LIN {X 0,Y 100.237,Z 319.477,A -85,B 0,C 180,E1 -28284.878,E2 -28284.878} C_VEL
LIN {X 0,Y 100.973,Z 322.725,A -85,B 0,C 180,E1 -28289.159,E2 -28289.159} C_VEL
LIN {X 0,Y 101.731,Z 327.087,A -85,B 0,C 180,E1 -28293.993,E2 -28293.993} C_VEL
LIN {X 0,Y 102.226,Z 331.393,A -85,B 0,C 180,E1 -28298.225,E2 -28298.225} C_VEL
LIN {X 0,Y 102.183,Z 334.397,A -85,B 0,C 180,E1 -28300.829,E2 -28300.829} C_VEL
LIN {X 0,Y 101.856,Z 336.169,A -85,B 0,C 180,E1 -28302.111,E2 -28302.111} C_VEL
LIN {X 0,Y 101.066,Z 337.874,A -85,B 0,C 180,E1 -28303.092,E2 -28303.092} C_VEL
LIN {X 0,Y 94.071,Z 347.385,A -85,B 0,C 180,E1 -28307.74,E2 -28307.74} C_VEL
LIN {X 0,Y 87.576,Z 355.164,A -85,B 0,C 180,E1 -28313.275,E2 -28313.275} C_VEL
LIN {X 0,Y 82.169,Z 361.026,A -85,B 0,C 180,E1 -28319.116,E2 -28319.116} C_VEL
LIN {X 0,Y 77.494,Z 365.857,A -85,B 0,C 180,E1 -28325.906,E2 -28325.906} C_VEL
LIN {X 0,Y 73.914,Z 369.582,A -85,B 0,C 180,E1 -28333.418,E2 -28333.418} C_VEL
LIN {X 0,Y 72.209,Z 371.5,A -85,B 0,C 180,E1 -28338.75,E2 -28338.75} C_VEL
LIN {X 0,Y 70.595,Z 372.917,A -85,B 0,C 180,E1 -28343.171,E2 -28343.171} C_VEL
LIN {X 0,Y 68.413,Z 374.026,A -85,B 0,C 180,E1 -28347.646,E2 -28347.646} C_VEL
LIN {X 0,Y 64.554,Z 375.318,A -85,B 0,C 180,E1 -28357.388,E2 -28357.388} C_VEL
LIN {X 0,Y 64.037,Z 375.526,A -85,B 0,C 180,E1 -28362.692,E2 -28362.692} C_VEL
LIN {X 0,Y 64.223,Z 375.507,A -85,B 0,C 180,E1 -28364.464,E2 -28364.464} C_VEL
LIN {X 0,Y 66.935,Z 374.948,A -85,B 0,C 180,E1 -28374.824,E2 -28374.824} C_VEL
LIN {X 0,Y 72.356,Z 372.767,A -85,B 0,C 180,E1 -28385.636,E2 -28385.636} C_VEL
LIN {X 0,Y 77.872,Z 370.014,A -85,B 0,C 180,E1 -28392.59,E2 -28392.59} C_VEL
LIN {X 0,Y 84.271,Z 366.237,A -85,B 0,C 180,E1 -28398.63,E2 -28398.63} C_VEL
LIN {X 0,Y 91.429,Z 361.324,A -85,B 0,C 180,E1 -28403.804,E2 -28403.804} C_VEL
LIN {X 0,Y 99.192,Z 355.123,A -85,B 0,C 180,E1 -28408.225,E2 -28408.225} C_VEL
LIN {X 0,Y 103.769,Z 350.924,A -85,B 0,C 180,E1 -28410.467,E2 -28410.467} C_VEL
LIN {X 0,Y 104.812,Z 347.909,A -85,B 0,C 180,E1 -28414.16,E2 -28414.16} C_VEL
LIN {X 0,Y 105.601,Z 344.619,A -85,B 0,C 180,E1 -28418.69,E2 -28418.69} C_VEL
LIN {X 0,Y 105.994,Z 341.263,A -85,B 0,C 180,E1 -28424.619,E2 -28424.619} C_VEL
LIN {X 0,Y 106.042,Z 339.662,A -85,B 0,C 180,E1 -28428.531,E2 -28428.531} C_VEL
LIN {X 0,Y 106.187,Z 338.276,A -85,B 0,C 180,E1 -28433.059,E2 -28433.059} C_VEL
LIN {X 0,Y 106.837,Z 336.92,A -85,B 0,C 180,E1 -28440,E2 -28440} C_VEL
LIN {X 0,Y 105.925,Z 338.695,A -85,B 0,C 180,E1 -28445.656,E2 -28445.656} C_VEL
LIN {X 0,Y 105.423,Z 341.22,A -85,B 0,C 180,E1 -28451.536,E2 -28451.536} C_VEL
LIN {X 0,Y 105.037,Z 343.497,A -85,B 0,C 180,E1 -28455.523,E2 -28455.523} C_VEL
LIN {X 0,Y 104.468,Z 346.468,A -85,B 0,C 180,E1 -28459.656,E2 -28459.656} C_VEL
LIN {X 0,Y 103.329,Z 351.55,A -85,B 0,C 180,E1 -28465.77,E2 -28465.77} C_VEL
LIN {X 0,Y 102.94,Z 353.062,A -85,B 0,C 180,E1 -28467.447,E2 -28467.447} C_VEL
LIN {X 0,Y 101.965,Z 354.793,A -85,B 0,C 180,E1 -28468.847,E2 -28468.847} C_VEL
LIN {X 0,Y 96.86,Z 361.172,A -85,B 0,C 180,E1 -28473.456,E2 -28473.456} C_VEL
LIN {X 0,Y 94.423,Z 363.454,A -85,B 0,C 180,E1 -28475.052,E2 -28475.052} C_VEL
LIN {X 0,Y 86.797,Z 369.418,A -85,B 0,C 180,E1 -28479.727,E2 -28479.727} C_VEL
LIN {X 0,Y 79.888,Z 374.149,A -85,B 0,C 180,E1 -28485.279,E2 -28485.279} C_VEL
LIN {X 0,Y 73.847,Z 377.783,A -85,B 0,C 180,E1 -28491.796,E2 -28491.796} C_VEL
LIN {X 0,Y 68.871,Z 380.421,A -85,B 0,C 180,E1 -28499.331,E2 -28499.331} C_VEL
LIN {X 0,Y 66.357,Z 381.688,A -85,B 0,C 180,E1 -28504.945,E2 -28504.945} C_VEL
LIN {X 0,Y 64.543,Z 382.528,A -85,B 0,C 180,E1 -28510.943,E2 -28510.943} C_VEL
LIN {X 0,Y 62.964,Z 383.019,A -85,B 0,C 180,E1 -28523.601,E2 -28523.601} C_VEL
LIN {X 0,Y 63.17,Z 382.685,A -85,B 0,C 180,E1 -28530.009,E2 -28530.009} C_VEL
LIN {X 0,Y 62.978,Z 381.865,A -85,B 0,C 180,E1 -28536.417,E2 -28536.417} C_VEL
LIN {X 0,Y 63.413,Z 380.607,A -85,B 0,C 180,E1 -28542.816,E2 -28542.816} C_VEL
LIN {X 0,Y 65.37,Z 377.946,A -85,B 0,C 180,E1 -28552.114,E2 -28552.114} C_VEL
LIN {X 0,Y 68.839,Z 374.259,A -85,B 0,C 180,E1 -28560.704,E2 -28560.704} C_VEL
LIN {X 0,Y 73.698,Z 369.456,A -85,B 0,C 180,E1 -28568.316,E2 -28568.316} C_VEL
LIN {X 0,Y 79.495,Z 363.369,A -85,B 0,C 180,E1 -28575.023,E2 -28575.023} C_VEL
LIN {X 0,Y 85.266,Z 357.204,A -85,B 0,C 180,E1 -28579.689,E2 -28579.689} C_VEL
LIN {X 0,Y 88.32,Z 352.824,A -85,B 0,C 180,E1 -28582.736,E2 -28582.736} C_VEL
LIN {X 0,Y 93.291,Z 344.019,A -85,B 0,C 180,E1 -28588.175,E2 -28588.175} C_VEL
LIN {X 0,Y 95.208,Z 339.981,A -85,B 0,C 180,E1 -28590.414,E2 -28590.414} C_VEL
LIN {X 0,Y 95.71,Z 338.033,A -85,B 0,C 180,E1 -28591.796,E2 -28591.796} C_VEL
LIN {X 0,Y 95.932,Z 333.079,A -85,B 0,C 180,E1 -28596.239,E2 -28596.239} C_VEL
LIN {X 0,Y 95.806,Z 327.088,A -85,B 0,C 180,E1 -28602.504,E2 -28602.504} C_VEL
LIN {X 0,Y 95.602,Z 323.433,A -85,B 0,C 180,E1 -28607.26,E2 -28607.26} C_VEL
LIN {X 0,Y 95.363,Z 320.851,A -85,B 0,C 180,E1 -28611.524,E2 -28611.524} C_VEL
LIN {X 0,Y 95.158,Z 319.066,A -85,B 0,C 180,E1 -28615.765,E2 -28615.765} C_VEL
LIN {X 0,Y 94.982,Z 318.072,A -85,B 0,C 180,E1 -28620.001,E2 -28620.001} C_VEL
LIN {X 0,Y 94.554,Z 318.54,A -85,B 0,C 180,E1 -28627.291,E2 -28627.291} C_VEL
LIN {X 0,Y 94.796,Z 319.647,A -85,B 0,C 180,E1 -28632.851,E2 -28632.851} C_VEL
LIN {X 0,Y 95.306,Z 322.239,A -85,B 0,C 180,E1 -28639.381,E2 -28639.381} C_VEL
LIN {X 0,Y 95.804,Z 324.716,A -85,B 0,C 180,E1 -28643.814,E2 -28643.814} C_VEL
LIN {X 0,Y 96.283,Z 328.257,A -85,B 0,C 180,E1 -28648.835,E2 -28648.835} C_VEL
LIN {X 0,Y 96.701,Z 332.759,A -85,B 0,C 180,E1 -28654.231,E2 -28654.231} C_VEL
LIN {X 0,Y 96.706,Z 336.521,A -85,B 0,C 180,E1 -28658.149,E2 -28658.149} C_VEL
LIN {X 0,Y 96.26,Z 338.595,A -85,B 0,C 180,E1 -28659.941,E2 -28659.941} C_VEL
LIN {X 0,Y 91.388,Z 345.102,A -85,B 0,C 180,E1 -28663.056,E2 -28663.056} C_VEL
LIN {X 0,Y 84.354,Z 353.212,A -85,B 0,C 180,E1 -28668.191,E2 -28668.191} C_VEL
LIN {X 0,Y 78.146,Z 359.73,A -85,B 0,C 180,E1 -28674.218,E2 -28674.218} C_VEL
LIN {X 0,Y 72.707,Z 364.935,A -85,B 0,C 180,E1 -28681.089,E2 -28681.089} C_VEL
LIN {X 0,Y 68.382,Z 368.985,A -85,B 0,C 180,E1 -28688.908,E2 -28688.908} C_VEL
LIN {X 0,Y 65.282,Z 372.001,A -85,B 0,C 180,E1 -28697.557,E2 -28697.557} C_VEL
LIN {X 0,Y 64.053,Z 373.495,A -85,B 0,C 180,E1 -28703.692,E2 -28703.692} C_VEL
LIN {X 0,Y 63.432,Z 375.223,A -85,B 0,C 180,E1 -28716.352,E2 -28716.352} C_VEL
LIN {X 0,Y 64.223,Z 375.507,A -85,B 0,C 180,E1 -28724.464,E2 -28724.464} C_VEL
LIN {X 0,Y 64.648,Z 375.451,A -85,B 0,C 180,E1 -28729.706,E2 -28729.706} C_VEL
LIN {X 0,Y 64.641,Z 374.849,A -85,B 0,C 180,E1 -28738.499,E2 -28738.499} C_VEL
LIN {X 0,Y 66.024,Z 373.597,A -85,B 0,C 180,E1 -28747.062,E2 -28747.062} C_VEL
LIN {X 0,Y 68.47,Z 372.339,A -85,B 0,C 180,E1 -28751.532,E2 -28751.532} C_VEL
LIN {X 0,Y 75.001,Z 369.204,A -85,B 0,C 180,E1 -28758.547,E2 -28758.547} C_VEL
LIN {X 0,Y 82.221,Z 365.031,A -85,B 0,C 180,E1 -28764.282,E2 -28764.282} C_VEL
LIN {X 0,Y 91.461,Z 358.667,A -85,B 0,C 180,E1 -28769.808,E2 -28769.808} C_VEL
LIN {X 0,Y 98.395,Z 352.93,A -85,B 0,C 180,E1 -28773.236,E2 -28773.236} C_VEL
LIN {X 0,Y 99.401,Z 350.464,A -85,B 0,C 180,E1 -28776.785,E2 -28776.785} C_VEL
LIN {X 0,Y 99.974,Z 348.824,A -85,B 0,C 180,E1 -28779.421,E2 -28779.421} C_VEL
LIN {X 0,Y 100.492,Z 346.577,A -85,B 0,C 180,E1 -28783.755,E2 -28783.755} C_VEL
LIN {X 0,Y 100.801,Z 344.873,A -85,B 0,C 180,E1 -28787.926,E2 -28787.926} C_VEL
LIN {X 0,Y 101.047,Z 343.664,A -85,B 0,C 180,E1 -28792.003,E2 -28792.003} C_VEL
LIN {X 0,Y 101.898,Z 342.177,A -85,B 0,C 180,E1 -28800,E2 -28800} C_VEL
LIN {X 0,Y 101.178,Z 343.307,A -85,B 0,C 180,E1 -28803.983,E2 -28803.983} C_VEL
LIN {X 0,Y 100.228,Z 346.059,A -85,B 0,C 180,E1 -28811.016,E2 -28811.016} C_VEL
LIN {X 0,Y 99.786,Z 347.751,A -85,B 0,C 180,E1 -28814.271,E2 -28814.271} C_VEL
LIN {X 0,Y 98.749,Z 351.134,A -85,B 0,C 180,E1 -28819.418,E2 -28819.418} C_VEL
LIN {X 0,Y 97.855,Z 354.006,A -85,B 0,C 180,E1 -28823.264,E2 -28823.264} C_VEL
LIN {X 0,Y 97.097,Z 355.997,A -85,B 0,C 180,E1 -28825.74,E2 -28825.74} C_VEL
LIN {X 0,Y 94.026,Z 359.653,A -85,B 0,C 180,E1 -28828.581,E2 -28828.581} C_VEL
LIN {X 0,Y 90.515,Z 363.192,A -85,B 0,C 180,E1 -28831.353,E2 -28831.353} C_VEL
LIN {X 0,Y 82.412,Z 369.123,A -85,B 0,C 180,E1 -28835.902,E2 -28835.902} C_VEL
LIN {X 0,Y 74.979,Z 373.826,A -85,B 0,C 180,E1 -28841.434,E2 -28841.434} C_VEL
LIN {X 0,Y 68.372,Z 377.433,A -85,B 0,C 180,E1 -28848.089,E2 -28848.089} C_VEL
LIN {X 0,Y 62.849,Z 380.046,A -85,B 0,C 180,E1 -28856.017,E2 -28856.017} C_VEL
LIN {X 0,Y 59.956,Z 381.297,A -85,B 0,C 180,E1 -28862.05,E2 -28862.05} C_VEL
LIN {X 0,Y 57.848,Z 382.116,A -85,B 0,C 180,E1 -28868.636,E2 -28868.636} C_VEL
LIN {X 0,Y 55.902,Z 382.584,A -85,B 0,C 180,E1 -28882.788,E2 -28882.788} C_VEL
LIN {X 0,Y 56.072,Z 382.239,A -85,B 0,C 180,E1 -28890.011,E2 -28890.011} C_VEL
LIN {X 0,Y 55.913,Z 381.394,A -85,B 0,C 180,E1 -28897.232,E2 -28897.232} C_VEL
LIN {X 0,Y 56.479,Z 380.123,A -85,B 0,C 180,E1 -28904.421,E2 -28904.421} C_VEL
LIN {X 0,Y 58.799,Z 377.435,A -85,B 0,C 180,E1 -28914.741,E2 -28914.741} C_VEL
LIN {X 0,Y 62.82,Z 373.723,A -85,B 0,C 180,E1 -28924.024,E2 -28924.024} C_VEL
LIN {X 0,Y 68.232,Z 368.889,A -85,B 0,C 180,E1 -28932.041,E2 -28932.041} C_VEL
LIN {X 0,Y 74.64,Z 362.773,A -85,B 0,C 180,E1 -28938.886,E2 -28938.886} C_VEL
LIN {X 0,Y 80.783,Z 356.563,A -85,B 0,C 180,E1 -28943.597,E2 -28943.597} C_VEL
LIN {X 0,Y 86.082,Z 348.868,A -85,B 0,C 180,E1 -28949.022,E2 -28949.022} C_VEL
LIN {X 0,Y 89.62,Z 342.86,A -85,B 0,C 180,E1 -28952.689,E2 -28952.689} C_VEL
LIN {X 0,Y 90.054,Z 341.88,A -85,B 0,C 180,E1 -28953.336,E2 -28953.336} C_VEL
LIN {X 0,Y 90.717,Z 337.829,A -85,B 0,C 180,E1 -28957.21,E2 -28957.21} C_VEL
LIN {X 0,Y 91.045,Z 333.492,A -85,B 0,C 180,E1 -28962.015,E2 -28962.015} C_VEL
LIN {X 0,Y 91.158,Z 329.964,A -85,B 0,C 180,E1 -28966.627,E2 -28966.627} C_VEL
LIN {X 0,Y 91.222,Z 327.208,A -85,B 0,C 180,E1 -28971.137,E2 -28971.137} C_VEL
LIN {X 0,Y 91.206,Z 325.221,A -85,B 0,C 180,E1 -28975.581,E2 -28975.581} C_VEL
LIN {X 0,Y 91.138,Z 324.105,A -85,B 0,C 180,E1 -28980.001,E2 -28980.001} C_VEL
LIN {X 0,Y 90.793,Z 324.195,A -85,B 0,C 180,E1 -28984.44,E2 -28984.44} C_VEL
LIN {X 0,Y 90.699,Z 324.724,A -85,B 0,C 180,E1 -28988.916,E2 -28988.916} C_VEL
LIN {X 0,Y 90.788,Z 325.793,A -85,B 0,C 180,E1 -28993.429,E2 -28993.429} C_VEL
LIN {X 0,Y 91.017,Z 328.575,A -85,B 0,C 180,E1 -29000.336,E2 -29000.336} C_VEL
LIN {X 0,Y 91.214,Z 331.227,A -85,B 0,C 180,E1 -29005.074,E2 -29005.074} C_VEL
LIN {X 0,Y 91.32,Z 335.045,A -85,B 0,C 180,E1 -29010.563,E2 -29010.563} C_VEL
LIN {X 0,Y 91.214,Z 338.829,A -85,B 0,C 180,E1 -29015.27,E2 -29015.27} C_VEL
LIN {X 0,Y 91.092,Z 339.907,A -85,B 0,C 180,E1 -29016.461,E2 -29016.461} C_VEL
LIN {X 0,Y 90.483,Z 341.271,A -85,B 0,C 180,E1 -29017.51,E2 -29017.51} C_VEL
LIN {X 0,Y 82.883,Z 350.012,A -85,B 0,C 180,E1 -29022.092,E2 -29022.092} C_VEL
LIN {X 0,Y 75.821,Z 357.245,A -85,B 0,C 180,E1 -29027.767,E2 -29027.767} C_VEL
LIN {X 0,Y 69.311,Z 363.196,A -85,B 0,C 180,E1 -29034.618,E2 -29034.618} C_VEL
LIN {X 0,Y 63.233,Z 368.281,A -85,B 0,C 180,E1 -29043.594,E2 -29043.594} C_VEL
LIN {X 0,Y 60.492,Z 370.6,A -85,B 0,C 180,E1 -29049.592,E2 -29049.592} C_VEL
LIN {X 0,Y 58.396,Z 372.497,A -85,B 0,C 180,E1 -29056.062,E2 -29056.062} C_VEL
LIN {X 0,Y 57.029,Z 373.968,A -85,B 0,C 180,E1 -29062.911,E2 -29062.911} C_VEL
LIN {X 0,Y 56.29,Z 375.318,A -85,B 0,C 180,E1 -29072.759,E2 -29072.759} C_VEL
LIN {X 0,Y 57.233,Z 375.947,A -85,B 0,C 180,E1 -29085.462,E2 -29085.462} C_VEL
LIN {X 0,Y 60.535,Z 375.346,A -85,B 0,C 180,E1 -29097.66,E2 -29097.66} C_VEL
LIN {X 0,Y 66.699,Z 373.139,A -85,B 0,C 180,E1 -29109.202,E2 -29109.202} C_VEL
LIN {X 0,Y 68.47,Z 372.339,A -85,B 0,C 180,E1 -29111.532,E2 -29111.532} C_VEL
LIN {X 0,Y 71.248,Z 370.931,A -85,B 0,C 180,E1 -29115.639,E2 -29115.639} C_VEL
LIN {X 0,Y 74.981,Z 368.205,A -85,B 0,C 180,E1 -29122.527,E2 -29122.527} C_VEL
LIN {X 0,Y 78.416,Z 365.56,A -85,B 0,C 180,E1 -29127.52,E2 -29127.52} C_VEL
LIN {X 0,Y 81.823,Z 363.199,A -85,B 0,C 180,E1 -29130.543,E2 -29130.543} C_VEL
LIN {X 0,Y 83.165,Z 362.307,A -85,B 0,C 180,E1 -29131.348,E2 -29131.348} C_VEL
LIN {X 0,Y 92.483,Z 355.615,A -85,B 0,C 180,E1 -29135.754,E2 -29135.754} C_VEL
LIN {X 0,Y 93.56,Z 354.037,A -85,B 0,C 180,E1 -29137.939,E2 -29137.939} C_VEL
LIN {X 0,Y 94.243,Z 352.683,A -85,B 0,C 180,E1 -29140.392,E2 -29140.392} C_VEL
LIN {X 0,Y 94.887,Z 350.88,A -85,B 0,C 180,E1 -29144.314,E2 -29144.314} C_VEL
LIN {X 0,Y 95.225,Z 349.837,A -85,B 0,C 180,E1 -29147.207,E2 -29147.207} C_VEL
LIN {X 0,Y 95.624,Z 348.576,A -85,B 0,C 180,E1 -29151.547,E2 -29151.547} C_VEL
LIN {X 0,Y 96.107,Z 347.703,A -85,B 0,C 180,E1 -29155.806,E2 -29155.806} C_VEL
LIN {X 0,Y 96.662,Z 347.171,A -85,B 0,C 180,E1 -29159.999,E2 -29159.999} C_VEL
LIN {X 0,Y 95.814,Z 348.347,A -85,B 0,C 180,E1 -29164.206,E2 -29164.206} C_VEL
LIN {X 0,Y 95.056,Z 349.853,A -85,B 0,C 180,E1 -29168.503,E2 -29168.503} C_VEL
LIN {X 0,Y 94.126,Z 352.35,A -85,B 0,C 180,E1 -29173.941,E2 -29173.941} C_VEL
LIN {X 0,Y 92.564,Z 356.027,A -85,B 0,C 180,E1 -29179.978,E2 -29179.978} C_VEL
LIN {X 0,Y 91.183,Z 358.775,A -85,B 0,C 180,E1 -29183.814,E2 -29183.814} C_VEL
LIN {X 0,Y 86.9,Z 362.921,A -85,B 0,C 180,E1 -29187.191,E2 -29187.191} C_VEL
LIN {X 0,Y 81.237,Z 366.997,A -85,B 0,C 180,E1 -29190.119,E2 -29190.119} C_VEL
LIN {X 0,Y 72.279,Z 372.475,A -85,B 0,C 180,E1 -29195.69,E2 -29195.69} C_VEL
LIN {X 0,Y 63.239,Z 377.083,A -85,B 0,C 180,E1 -29203.764,E2 -29203.764} C_VEL
LIN {X 0,Y 57.085,Z 379.672,A -85,B 0,C 180,E1 -29212.02,E2 -29212.02} C_VEL
LIN {X 0,Y 53.748,Z 380.902,A -85,B 0,C 180,E1 -29218.477,E2 -29218.477} C_VEL
LIN {X 0,Y 51.279,Z 381.705,A -85,B 0,C 180,E1 -29225.735,E2 -29225.735} C_VEL
LIN {X 0,Y 48.842,Z 382.149,A -85,B 0,C 180,E1 -29241.739,E2 -29241.739} C_VEL
LIN {X 0,Y 48.957,Z 381.791,A -85,B 0,C 180,E1 -29250.012,E2 -29250.012} C_VEL
LIN {X 0,Y 48.852,Z 380.923,A -85,B 0,C 180,E1 -29258.284,E2 -29258.284} C_VEL
LIN {X 0,Y 51.265,Z 377.948,A -85,B 0,C 180,E1 -29274.297,E2 -29274.297} C_VEL
LIN {X 0,Y 55.307,Z 374.554,A -85,B 0,C 180,E1 -29284.891,E2 -29284.891} C_VEL
LIN {X 0,Y 60.94,Z 370.081,A -85,B 0,C 180,E1 -29293.798,E2 -29293.798} C_VEL
LIN {X 0,Y 68.583,Z 363.553,A -85,B 0,C 180,E1 -29302.06,E2 -29302.06} C_VEL
LIN {X 0,Y 75.419,Z 357.302,A -85,B 0,C 180,E1 -29307.014,E2 -29307.014} C_VEL
LIN {X 0,Y 81.128,Z 349.972,A -85,B 0,C 180,E1 -29312.43,E2 -29312.43} C_VEL
LIN {X 0,Y 84.715,Z 344.564,A -85,B 0,C 180,E1 -29315.878,E2 -29315.878} C_VEL
LIN {X 0,Y 85.533,Z 341.107,A -85,B 0,C 180,E1 -29319.655,E2 -29319.655} C_VEL
LIN {X 0,Y 86.334,Z 336.244,A -85,B 0,C 180,E1 -29325.865,E2 -29325.865} C_VEL
LIN {X 0,Y 86.697,Z 333.277,A -85,B 0,C 180,E1 -29330.67,E2 -29330.67} C_VEL
LIN {X 0,Y 86.872,Z 331.211,A -85,B 0,C 180,E1 -29335.36,E2 -29335.36} C_VEL
LIN {X 0,Y 86.972,Z 329.919,A -85,B 0,C 180,E1 -29340.001,E2 -29340.001} C_VEL
LIN {X 0,Y 86.62,Z 329.987,A -85,B 0,C 180,E1 -29344.654,E2 -29344.654} C_VEL
LIN {X 0,Y 86.437,Z 330.595,A -85,B 0,C 180,E1 -29349.359,E2 -29349.359} C_VEL
LIN {X 0,Y 86.351,Z 331.74,A -85,B 0,C 180,E1 -29354.133,E2 -29354.133} C_VEL
LIN {X 0,Y 86.344,Z 333.539,A -85,B 0,C 180,E1 -29359.001,E2 -29359.001} C_VEL
LIN {X 0,Y 86.249,Z 336.059,A -85,B 0,C 180,E1 -29364.044,E2 -29364.044} C_VEL
LIN {X 0,Y 86.019,Z 339.367,A -85,B 0,C 180,E1 -29369.356,E2 -29369.356} C_VEL
LIN {X 0,Y 85.806,Z 341.512,A -85,B 0,C 180,E1 -29372.382,E2 -29372.382} C_VEL
LIN {X 0,Y 85.18,Z 343.313,A -85,B 0,C 180,E1 -29374.392,E2 -29374.392} C_VEL
LIN {X 0,Y 77.02,Z 351.987,A -85,B 0,C 180,E1 -29379.127,E2 -29379.127} C_VEL
LIN {X 0,Y 69.522,Z 358.902,A -85,B 0,C 180,E1 -29384.946,E2 -29384.946} C_VEL
LIN {X 0,Y 62.043,Z 365.019,A -85,B 0,C 180,E1 -29392.951,E2 -29392.951} C_VEL
LIN {X 0,Y 55.418,Z 370.031,A -85,B 0,C 180,E1 -29403.637,E2 -29403.637} C_VEL
LIN {X 0,Y 51.563,Z 372.992,A -85,B 0,C 180,E1 -29414.169,E2 -29414.169} C_VEL
LIN {X 0,Y 50,Z 374.439,A -85,B 0,C 180,E1 -29421.908,E2 -29421.908} C_VEL
LIN {X 0,Y 49.222,Z 375.645,A -85,B 0,C 180,E1 -29431.827,E2 -29431.827} C_VEL
LIN {X 0,Y 50.174,Z 376.399,A -85,B 0,C 180,E1 -29446.256,E2 -29446.256} C_VEL
LIN {X 0,Y 51.858,Z 376.279,A -85,B 0,C 180,E1 -29453.977,E2 -29453.977} C_VEL
LIN {X 0,Y 57.486,Z 374.826,A -85,B 0,C 180,E1 -29467.669,E2 -29467.669} C_VEL
LIN {X 0,Y 62.798,Z 372.906,A -85,B 0,C 180,E1 -29475.214,E2 -29475.214} C_VEL
LIN {X 0,Y 70.489,Z 369.536,A -85,B 0,C 180,E1 -29482.89,E2 -29482.89} C_VEL
LIN {X 0,Y 78.277,Z 365.334,A -85,B 0,C 180,E1 -29488.518,E2 -29488.518} C_VEL
LIN {X 0,Y 83.165,Z 362.307,A -85,B 0,C 180,E1 -29491.348,E2 -29491.348} C_VEL
LIN {X 0,Y 85.444,Z 360.629,A -85,B 0,C 180,E1 -29493.102,E2 -29493.102} C_VEL
LIN {X 0,Y 86.983,Z 359.119,A -85,B 0,C 180,E1 -29495.237,E2 -29495.237} C_VEL
LIN {X 0,Y 88.325,Z 357.205,A -85,B 0,C 180,E1 -29498.812,E2 -29498.812} C_VEL
LIN {X 0,Y 88.923,Z 355.658,A -85,B 0,C 180,E1 -29502.736,E2 -29502.736} C_VEL
LIN {X 0,Y 89.887,Z 353.242,A -85,B 0,C 180,E1 -29510.873,E2 -29510.873} C_VEL
LIN {X 0,Y 90.522,Z 352.31,A -85,B 0,C 180,E1 -29515.547,E2 -29515.547} C_VEL
LIN {X 0,Y 91.099,Z 351.87,A -85,B 0,C 180,E1 -29519.999,E2 -29519.999} C_VEL
LIN {X 0,Y 90.114,Z 353.06,A -85,B 0,C 180,E1 -29524.473,E2 -29524.473} C_VEL
LIN {X 0,Y 88.8,Z 355.546,A -85,B 0,C 180,E1 -29531.411,E2 -29531.411} C_VEL
LIN {X 0,Y 87.594,Z 357.693,A -85,B 0,C 180,E1 -29535.702,E2 -29535.702} C_VEL
LIN {X 0,Y 85.976,Z 360.499,A -85,B 0,C 180,E1 -29540.469,E2 -29540.469} C_VEL
LIN {X 0,Y 84.92,Z 361.58,A -85,B 0,C 180,E1 -29541.662,E2 -29541.662} C_VEL
LIN {X 0,Y 82.379,Z 363.724,A -85,B 0,C 180,E1 -29543.511,E2 -29543.511} C_VEL
LIN {X 0,Y 72.036,Z 370.183,A -85,B 0,C 180,E1 -29548.609,E2 -29548.609} C_VEL
LIN {X 0,Y 63.708,Z 374.454,A -85,B 0,C 180,E1 -29554.188,E2 -29554.188} C_VEL
LIN {X 0,Y 56.12,Z 377.674,A -85,B 0,C 180,E1 -29561.305,E2 -29561.305} C_VEL
LIN {X 0,Y 51.661,Z 379.298,A -85,B 0,C 180,E1 -29567.156,E2 -29567.156} C_VEL
LIN {X 0,Y 47.805,Z 380.505,A -85,B 0,C 180,E1 -29573.996,E2 -29573.996} C_VEL
LIN {X 0,Y 42.815,Z 381.695,A -85,B 0,C 180,E1 -29590.849,E2 -29590.849} C_VEL
LIN {X 0,Y 41.826,Z 381.715,A -85,B 0,C 180,E1 -29600.341,E2 -29600.341} C_VEL
LIN {X 0,Y 41.846,Z 381.34,A -85,B 0,C 180,E1 -29610.014,E2 -29610.014} C_VEL
LIN {X 0,Y 41.814,Z 380.452,A -85,B 0,C 180,E1 -29619.69,E2 -29619.69} C_VEL
LIN {X 0,Y 42.805,Z 379.155,A -85,B 0,C 180,E1 -29629.184,E2 -29629.184} C_VEL
LIN {X 0,Y 46.21,Z 376.414,A -85,B 0,C 180,E1 -29642.176,E2 -29642.176} C_VEL
LIN {X 0,Y 51.604,Z 372.649,A -85,B 0,C 180,E1 -29652.933,E2 -29652.933} C_VEL
LIN {X 0,Y 58.38,Z 367.753,A -85,B 0,C 180,E1 -29661.505,E2 -29661.505} C_VEL
LIN {X 0,Y 63.845,Z 363.455,A -85,B 0,C 180,E1 -29666.606,E2 -29666.606} C_VEL
LIN {X 0,Y 70.36,Z 357.96,A -85,B 0,C 180,E1 -29670.944,E2 -29670.944} C_VEL
LIN {X 0,Y 75.426,Z 352.294,A -85,B 0,C 180,E1 -29675.314,E2 -29675.314} C_VEL
LIN {X 0,Y 78.492,Z 348.429,A -85,B 0,C 180,E1 -29677.964,E2 -29677.964} C_VEL
LIN {X 0,Y 79.633,Z 346.687,A -85,B 0,C 180,E1 -29679.328,E2 -29679.328} C_VEL
LIN {X 0,Y 80.895,Z 342.446,A -85,B 0,C 180,E1 -29684.893,E2 -29684.893} C_VEL
LIN {X 0,Y 81.661,Z 339.238,A -85,B 0,C 180,E1 -29690.089,E2 -29690.089} C_VEL
LIN {X 0,Y 81.998,Z 337.91,A -85,B 0,C 180,E1 -29692.614,E2 -29692.614} C_VEL
LIN {X 0,Y 82.202,Z 336.906,A -85,B 0,C 180,E1 -29695.096,E2 -29695.096} C_VEL
LIN {X 0,Y 82.468,Z 335.527,A -85,B 0,C 180,E1 -29700.001,E2 -29700.001} C_VEL
LIN {X 0,Y 82.118,Z 335.554,A -85,B 0,C 180,E1 -29704.91,E2 -29704.91} C_VEL
LIN {X 0,Y 81.823,Z 336.18,A -85,B 0,C 180,E1 -29709.892,E2 -29709.892} C_VEL
LIN {X 0,Y 81.538,Z 337.5,A -85,B 0,C 180,E1 -29714.986,E2 -29714.986} C_VEL
LIN {X 0,Y 81.331,Z 339.396,A -85,B 0,C 180,E1 -29720.222,E2 -29720.222} C_VEL
LIN {X 0,Y 80.892,Z 342.18,A -85,B 0,C 180,E1 -29725.748,E2 -29725.748} C_VEL
LIN {X 0,Y 80.464,Z 344.172,A -85,B 0,C 180,E1 -29729.125,E2 -29729.125} C_VEL
LIN {X 0,Y 79.921,Z 345.594,A -85,B 0,C 180,E1 -29730.962,E2 -29730.962} C_VEL
LIN {X 0,Y 71.367,Z 353.845,A -85,B 0,C 180,E1 -29735.652,E2 -29735.652} C_VEL
LIN {X 0,Y 62.762,Z 361.027,A -85,B 0,C 180,E1 -29742.213,E2 -29742.213} C_VEL
LIN {X 0,Y 55.113,Z 366.582,A -85,B 0,C 180,E1 -29750.373,E2 -29750.373} C_VEL
LIN {X 0,Y 49.183,Z 370.549,A -85,B 0,C 180,E1 -29759.977,E2 -29759.977} C_VEL
LIN {X 0,Y 44.804,Z 373.488,A -85,B 0,C 180,E1 -29771.702,E2 -29771.702} C_VEL
LIN {X 0,Y 42.993,Z 374.91,A -85,B 0,C 180,E1 -29780.578,E2 -29780.578} C_VEL
LIN {X 0,Y 42.169,Z 375.923,A -85,B 0,C 180,E1 -29789.986,E2 -29789.986} C_VEL
LIN {X 0,Y 42.316,Z 376.563,A -85,B 0,C 180,E1 -29799.546,E2 -29799.546} C_VEL
LIN {X 0,Y 43.383,Z 376.834,A -85,B 0,C 180,E1 -29808.891,E2 -29808.891} C_VEL
LIN {X 0,Y 45.448,Z 376.688,A -85,B 0,C 180,E1 -29817.625,E2 -29817.625} C_VEL
LIN {X 0,Y 52.018,Z 375.212,A -85,B 0,C 180,E1 -29832.48,E2 -29832.48} C_VEL
LIN {X 0,Y 56.394,Z 373.882,A -85,B 0,C 180,E1 -29838.378,E2 -29838.378} C_VEL
LIN {X 0,Y 63.763,Z 371.054,A -85,B 0,C 180,E1 -29845.739,E2 -29845.739} C_VEL
LIN {X 0,Y 71.942,Z 367.191,A -85,B 0,C 180,E1 -29851.529,E2 -29851.529} C_VEL
LIN {X 0,Y 80.669,Z 362.187,A -85,B 0,C 180,E1 -29856.154,E2 -29856.154} C_VEL
LIN {X 0,Y 86.705,Z 358.105,A -85,B 0,C 180,E1 -29858.752,E2 -29858.752} C_VEL
LIN {X 0,Y 88.357,Z 356.334,A -85,B 0,C 180,E1 -29861.447,E2 -29861.447} C_VEL
LIN {X 0,Y 89.297,Z 354.465,A -85,B 0,C 180,E1 -29866.342,E2 -29866.342} C_VEL
LIN {X 0,Y 89.887,Z 353.242,A -85,B 0,C 180,E1 -29870.873,E2 -29870.873} C_VEL
LIN {X 0,Y 89.751,Z 353.086,A -85,B 0,C 180,E1 -29873.339,E2 -29873.339} C_VEL
LIN {X 0,Y 88.353,Z 353.964,A -85,B 0,C 180,E1 -29876.565,E2 -29876.565} C_VEL
LIN {X 0,Y 84.277,Z 357.288,A -85,B 0,C 180,E1 -29884.164,E2 -29884.164} C_VEL
LIN {X 0,Y 83.095,Z 359.053,A -85,B 0,C 180,E1 -29889.738,E2 -29889.738} C_VEL
LIN {X 0,Y 82.352,Z 360.102,A -85,B 0,C 180,E1 -29892.318,E2 -29892.318} C_VEL
LIN {X 0,Y 80.747,Z 362.323,A -85,B 0,C 180,E1 -29896.81,E2 -29896.81} C_VEL
LIN {X 0,Y 79.644,Z 363.428,A -85,B 0,C 180,E1 -29898.472,E2 -29898.472} C_VEL
LIN {X 0,Y 78.237,Z 364.468,A -85,B 0,C 180,E1 -29899.425,E2 -29899.425} C_VEL
LIN {X 0,Y 68.906,Z 369.876,A -85,B 0,C 180,E1 -29903.394,E2 -29903.394} C_VEL
LIN {X 0,Y 59.976,Z 374.117,A -85,B 0,C 180,E1 -29908.517,E2 -29908.517} C_VEL
LIN {X 0,Y 51.679,Z 377.311,A -85,B 0,C 180,E1 -29915.338,E2 -29915.338} C_VEL
LIN {X 0,Y 46.675,Z 378.922,A -85,B 0,C 180,E1 -29921.181,E2 -29921.181} C_VEL
LIN {X 0,Y 42.238,Z 380.106,A -85,B 0,C 180,E1 -29928.294,E2 -29928.294} C_VEL
LIN {X 0,Y 36.164,Z 381.272,A -85,B 0,C 180,E1 -29947.146,E2 -29947.146} C_VEL
LIN {X 0,Y 34.818,Z 381.28,A -85,B 0,C 180,E1 -29958.372,E2 -29958.372} C_VEL
LIN {X 0,Y 34.734,Z 380.885,A -85,B 0,C 180,E1 -29970.017,E2 -29970.017} C_VEL
LIN {X 0,Y 34.8,Z 379.98,A -85,B 0,C 180,E1 -29981.668,E2 -29981.668} C_VEL
LIN {X 0,Y 36.157,Z 378.672,A -85,B 0,C 180,E1 -29992.894,E2 -29992.894} C_VEL
LIN {X 0,Y 40.331,Z 375.902,A -85,B 0,C 180,E1 -30007.6,E2 -30007.6} C_VEL
LIN {X 0,Y 46.625,Z 372.11,A -85,B 0,C 180,E1 -30018.929,E2 -30018.929} C_VEL
LIN {X 0,Y 54.202,Z 367.183,A -85,B 0,C 180,E1 -30027.457,E2 -30027.457} C_VEL
LIN {X 0,Y 61.082,Z 362.205,A -85,B 0,C 180,E1 -30032.804,E2 -30032.804} C_VEL
LIN {X 0,Y 67.107,Z 357.326,A -85,B 0,C 180,E1 -30036.423,E2 -30036.423} C_VEL
LIN {X 0,Y 73.947,Z 350.029,A -85,B 0,C 180,E1 -30041.904,E2 -30041.904} C_VEL
LIN {X 0,Y 74.801,Z 348.548,A -85,B 0,C 180,E1 -30043.629,E2 -30043.629} C_VEL
LIN {X 0,Y 76.259,Z 344.931,A -85,B 0,C 180,E1 -30049.379,E2 -30049.379} C_VEL
LIN {X 0,Y 77.142,Z 342.358,A -85,B 0,C 180,E1 -30054.773,E2 -30054.773} C_VEL
LIN {X 0,Y 77.596,Z 340.88,A -85,B 0,C 180,E1 -30060.001,E2 -30060.001} C_VEL
LIN {X 0,Y 77.253,Z 340.856,A -85,B 0,C 180,E1 -30065.22,E2 -30065.22} C_VEL
LIN {X 0,Y 76.823,Z 341.585,A -85,B 0,C 180,E1 -30070.543,E2 -30070.543} C_VEL
LIN {X 0,Y 76.404,Z 342.987,A -85,B 0,C 180,E1 -30076.02,E2 -30076.02} C_VEL
LIN {X 0,Y 75.777,Z 345.207,A -85,B 0,C 180,E1 -30081.939,E2 -30081.939} C_VEL
LIN {X 0,Y 74.964,Z 347.731,A -85,B 0,C 180,E1 -30087.029,E2 -30087.029} C_VEL
LIN {X 0,Y 66.054,Z 355.675,A -85,B 0,C 180,E1 -30091.643,E2 -30091.643} C_VEL
LIN {X 0,Y 57.364,Z 362.239,A -85,B 0,C 180,E1 -30097.777,E2 -30097.777} C_VEL
LIN {X 0,Y 48.337,Z 368.025,A -85,B 0,C 180,E1 -30107.091,E2 -30107.091} C_VEL
LIN {X 0,Y 41.286,Z 372.125,A -85,B 0,C 180,E1 -30119.274,E2 -30119.274} C_VEL
LIN {X 0,Y 38.158,Z 373.98,A -85,B 0,C 180,E1 -30128.369,E2 -30128.369} C_VEL
LIN {X 0,Y 35.177,Z 376.201,A -85,B 0,C 180,E1 -30147.404,E2 -30147.404} C_VEL
LIN {X 0,Y 35.314,Z 377.01,A -85,B 0,C 180,E1 -30161.462,E2 -30161.462} C_VEL
LIN {X 0,Y 36.732,Z 377.266,A -85,B 0,C 180,E1 -30172.481,E2 -30172.481} C_VEL
LIN {X 0,Y 39.26,Z 377.1,A -85,B 0,C 180,E1 -30182.464,E2 -30182.464} C_VEL
LIN {X 0,Y 47.002,Z 375.598,A -85,B 0,C 180,E1 -30198.366,E2 -30198.366} C_VEL
LIN {X 0,Y 51.93,Z 374.253,A -85,B 0,C 180,E1 -30204.273,E2 -30204.273} C_VEL
LIN {X 0,Y 60.04,Z 371.402,A -85,B 0,C 180,E1 -30211.371,E2 -30211.371} C_VEL
LIN {X 0,Y 68.825,Z 367.512,A -85,B 0,C 180,E1 -30216.762,E2 -30216.762} C_VEL
LIN {X 0,Y 78.053,Z 362.474,A -85,B 0,C 180,E1 -30220.962,E2 -30220.962} C_VEL
LIN {X 0,Y 81.201,Z 360.486,A -85,B 0,C 180,E1 -30222.161,E2 -30222.161} C_VEL
LIN {X 0,Y 82.942,Z 358.856,A -85,B 0,C 180,E1 -30225.273,E2 -30225.273} C_VEL
LIN {X 0,Y 84.016,Z 357.315,A -85,B 0,C 180,E1 -30231.514,E2 -30231.514} C_VEL
LIN {X 0,Y 84.669,Z 356.62,A -85,B 0,C 180,E1 -30235.238,E2 -30235.238} C_VEL
LIN {X 0,Y 85.245,Z 356.246,A -85,B 0,C 180,E1 -30239.999,E2 -30239.999} C_VEL
LIN {X 0,Y 84.277,Z 357.288,A -85,B 0,C 180,E1 -30244.164,E2 -30244.164} C_VEL
LIN {X 0,Y 83.182,Z 358.437,A -85,B 0,C 180,E1 -30246.808,E2 -30246.808} C_VEL
LIN {X 0,Y 80.849,Z 360.52,A -85,B 0,C 180,E1 -30250.034,E2 -30250.034} C_VEL
LIN {X 0,Y 77.707,Z 363.005,A -85,B 0,C 180,E1 -30252.851,E2 -30252.851} C_VEL
LIN {X 0,Y 74.827,Z 364.974,A -85,B 0,C 180,E1 -30254.588,E2 -30254.588} C_VEL
LIN {X 0,Y 72.641,Z 366.252,A -85,B 0,C 180,E1 -30255.472,E2 -30255.472} C_VEL
LIN {X 0,Y 63.189,Z 371.087,A -85,B 0,C 180,E1 -30259.054,E2 -30259.054} C_VEL
LIN {X 0,Y 53.864,Z 374.946,A -85,B 0,C 180,E1 -30264.056,E2 -30264.056} C_VEL
LIN {X 0,Y 42.316,Z 378.547,A -85,B 0,C 180,E1 -30273.884,E2 -30273.884} C_VEL
LIN {X 0,Y 37.212,Z 379.706,A -85,B 0,C 180,E1 -30280.959,E2 -30280.959} C_VEL
LIN {X 0,Y 29.71,Z 380.848,A -85,B 0,C 180,E1 -30301.787,E2 -30301.787} C_VEL
LIN {X 0,Y 27.88,Z 380.845,A -85,B 0,C 180,E1 -30315.421,E2 -30315.421} C_VEL
LIN {X 0,Y 27.632,Z 380.429,A -85,B 0,C 180,E1 -30330.021,E2 -30330.021} C_VEL
LIN {X 0,Y 27.869,Z 379.508,A -85,B 0,C 180,E1 -30344.629,E2 -30344.629} C_VEL
LIN {X 0,Y 29.705,Z 378.186,A -85,B 0,C 180,E1 -30358.263,E2 -30358.263} C_VEL
LIN {X 0,Y 34.943,Z 375.391,A -85,B 0,C 180,E1 -30374.769,E2 -30374.769} C_VEL
LIN {X 0,Y 42.276,Z 371.572,A -85,B 0,C 180,E1 -30386.248,E2 -30386.248} C_VEL
LIN {X 0,Y 50.697,Z 366.611,A -85,B 0,C 180,E1 -30394.327,E2 -30394.327} C_VEL
LIN {X 0,Y 59.874,Z 360.382,A -85,B 0,C 180,E1 -30399.918,E2 -30399.918} C_VEL
LIN {X 0,Y 62.999,Z 357.96,A -85,B 0,C 180,E1 -30401.513,E2 -30401.513} C_VEL
LIN {X 0,Y 68.792,Z 352.548,A -85,B 0,C 180,E1 -30405.664,E2 -30405.664} C_VEL
LIN {X 0,Y 70.128,Z 350.546,A -85,B 0,C 180,E1 -30408.438,E2 -30408.438} C_VEL
LIN {X 0,Y 71.061,Z 348.878,A -85,B 0,C 180,E1 -30411.552,E2 -30411.552} C_VEL
LIN {X 0,Y 71.651,Z 347.642,A -85,B 0,C 180,E1 -30414.372,E2 -30414.372} C_VEL
LIN {X 0,Y 72.425,Z 345.937,A -85,B 0,C 180,E1 -30420.001,E2 -30420.001} C_VEL
LIN {X 0,Y 71.956,Z 346.019,A -85,B 0,C 180,E1 -30426.388,E2 -30426.388} C_VEL
LIN {X 0,Y 71.484,Z 346.754,A -85,B 0,C 180,E1 -30431.341,E2 -30431.341} C_VEL
LIN {X 0,Y 70.804,Z 348.242,A -85,B 0,C 180,E1 -30437.325,E2 -30437.325} C_VEL
LIN {X 0,Y 70.123,Z 349.844,A -85,B 0,C 180,E1 -30441.683,E2 -30441.683} C_VEL
LIN {X 0,Y 68.882,Z 351.205,A -85,B 0,C 180,E1 -30443.306,E2 -30443.306} C_VEL
LIN {X 0,Y 59.601,Z 358.531,A -85,B 0,C 180,E1 -30447.805,E2 -30447.805} C_VEL
LIN {X 0,Y 50.689,Z 364.421,A -85,B 0,C 180,E1 -30453.685,E2 -30453.685} C_VEL
LIN {X 0,Y 42.469,Z 369.073,A -85,B 0,C 180,E1 -30461.848,E2 -30461.848} C_VEL
LIN {X 0,Y 35.396,Z 372.632,A -85,B 0,C 180,E1 -30473.42,E2 -30473.42} C_VEL
LIN {X 0,Y 31.679,Z 374.47,A -85,B 0,C 180,E1 -30483.639,E2 -30483.639} C_VEL
LIN {X 0,Y 28.245,Z 376.526,A -85,B 0,C 180,E1 -30504.465,E2 -30504.465} C_VEL
LIN {X 0,Y 28.396,Z 377.456,A -85,B 0,C 180,E1 -30524.308,E2 -30524.308} C_VEL
LIN {X 0,Y 30.278,Z 377.696,A -85,B 0,C 180,E1 -30537.639,E2 -30537.639} C_VEL
LIN {X 0,Y 37.658,Z 376.94,A -85,B 0,C 180,E1 -30558.265,E2 -30558.265} C_VEL
LIN {X 0,Y 42.596,Z 375.985,A -85,B 0,C 180,E1 -30565.559,E2 -30565.559} C_VEL
LIN {X 0,Y 48.109,Z 374.621,A -85,B 0,C 180,E1 -30571.199,E2 -30571.199} C_VEL
LIN {X 0,Y 56.97,Z 371.746,A -85,B 0,C 180,E1 -30577.673,E2 -30577.673} C_VEL
LIN {X 0,Y 66.333,Z 367.83,A -85,B 0,C 180,E1 -30582.437,E2 -30582.437} C_VEL
LIN {X 0,Y 75.517,Z 363.045,A -85,B 0,C 180,E1 -30585.897,E2 -30585.897} C_VEL
LIN {X 0,Y 77.498,Z 361.526,A -85,B 0,C 180,E1 -30589.55,E2 -30589.55} C_VEL
LIN {X 0,Y 78.538,Z 360.629,A -85,B 0,C 180,E1 -30594.865,E2 -30594.865} C_VEL
LIN {X 0,Y 79.182,Z 360.276,A -85,B 0,C 180,E1 -30599.999,E2 -30599.999} C_VEL
LIN {X 0,Y 77.691,Z 361.741,A -85,B 0,C 180,E1 -30605.774,E2 -30605.774} C_VEL
LIN {X 0,Y 76.433,Z 363.23,A -85,B 0,C 180,E1 -30610.596,E2 -30610.596} C_VEL
LIN {X 0,Y 74.965,Z 364.841,A -85,B 0,C 180,E1 -30614.331,E2 -30614.331} C_VEL
LIN {X 0,Y 72.641,Z 366.252,A -85,B 0,C 180,E1 -30615.472,E2 -30615.472} C_VEL
LIN {X 0,Y 67.518,Z 368.883,A -85,B 0,C 180,E1 -30616.65,E2 -30616.65} C_VEL
LIN {X 0,Y 58.348,Z 372.548,A -85,B 0,C 180,E1 -30617.493,E2 -30617.493} C_VEL
LIN {X 0,Y 48.961,Z 375.505,A -85,B 0,C 180,E1 -30618.791,E2 -30618.791} C_VEL
LIN {X 0,Y 43.584,Z 376.933,A -85,B 0,C 180,E1 -30621.246,E2 -30621.246} C_VEL
LIN {X 0,Y 32.975,Z 379.307,A -85,B 0,C 180,E1 -30631.548,E2 -30631.548} C_VEL
LIN {X 0,Y 23.667,Z 380.424,A -85,B 0,C 180,E1 -30653.596,E2 -30653.596} C_VEL
LIN {X 0,Y 21.079,Z 380.411,A -85,B 0,C 180,E1 -30670.554,E2 -30670.554} C_VEL
LIN {X 0,Y 20.522,Z 379.97,A -85,B 0,C 180,E1 -30690.029,E2 -30690.029} C_VEL
LIN {X 0,Y 21.051,Z 379.037,A -85,B 0,C 180,E1 -30709.533,E2 -30709.533} C_VEL
LIN {X 0,Y 23.666,Z 377.702,A -85,B 0,C 180,E1 -30726.467,E2 -30726.467} C_VEL
LIN {X 0,Y 30.295,Z 374.88,A -85,B 0,C 180,E1 -30744.32,E2 -30744.32} C_VEL
LIN {X 0,Y 38.765,Z 371.033,A -85,B 0,C 180,E1 -30755.061,E2 -30755.061} C_VEL
LIN {X 0,Y 48.022,Z 366.04,A -85,B 0,C 180,E1 -30762.08,E2 -30762.08} C_VEL
LIN {X 0,Y 57.814,Z 359.783,A -85,B 0,C 180,E1 -30766.574,E2 -30766.574} C_VEL
LIN {X 0,Y 61.038,Z 357.313,A -85,B 0,C 180,E1 -30768.199,E2 -30768.199} C_VEL
LIN {X 0,Y 64.203,Z 354.623,A -85,B 0,C 180,E1 -30770.176,E2 -30770.176} C_VEL
LIN {X 0,Y 65.724,Z 352.671,A -85,B 0,C 180,E1 -30773.862,E2 -30773.862} C_VEL
LIN {X 0,Y 66.889,Z 350.782,A -85,B 0,C 180,E1 -30780.001,E2 -30780.001} C_VEL
LIN {X 0,Y 66.597,Z 350.692,A -85,B 0,C 180,E1 -30786.058,E2 -30786.058} C_VEL
LIN {X 0,Y 65.404,Z 352.158,A -85,B 0,C 180,E1 -30794.706,E2 -30794.706} C_VEL
LIN {X 0,Y 65.319,Z 352.34,A -85,B 0,C 180,E1 -30795.602,E2 -30795.602} C_VEL
LIN {X 0,Y 64.355,Z 353.512,A -85,B 0,C 180,E1 -30798.393,E2 -30798.393} C_VEL
LIN {X 0,Y 55.049,Z 360.219,A -85,B 0,C 180,E1 -30802.215,E2 -30802.215} C_VEL
LIN {X 0,Y 44.395,Z 366.476,A -85,B 0,C 180,E1 -30808.5,E2 -30808.5} C_VEL
LIN {X 0,Y 33.818,Z 371.549,A -85,B 0,C 180,E1 -30819.142,E2 -30819.142} C_VEL
LIN {X 0,Y 25.524,Z 374.956,A -85,B 0,C 180,E1 -30836.558,E2 -30836.558} C_VEL
LIN {X 0,Y 21.523,Z 376.753,A -85,B 0,C 180,E1 -30858.425,E2 -30858.425} C_VEL
LIN {X 0,Y 21.586,Z 377.902,A -85,B 0,C 180,E1 -30888.972,E2 -30888.972} C_VEL
LIN {X 0,Y 24.192,Z 378.123,A -85,B 0,C 180,E1 -30905.492,E2 -30905.492} C_VEL
LIN {X 0,Y 33.333,Z 377.339,A -85,B 0,C 180,E1 -30927.463,E2 -30927.463} C_VEL
LIN {X 0,Y 39.006,Z 376.371,A -85,B 0,C 180,E1 -30934.238,E2 -30934.238} C_VEL
LIN {X 0,Y 45.105,Z 374.985,A -85,B 0,C 180,E1 -30939.173,E2 -30939.173} C_VEL
LIN {X 0,Y 57.558,Z 371.008,A -85,B 0,C 180,E1 -30945.864,E2 -30945.864} C_VEL
LIN {X 0,Y 67.884,Z 366.554,A -85,B 0,C 180,E1 -30949.535,E2 -30949.535} C_VEL
LIN {X 0,Y 71.173,Z 364.869,A -85,B 0,C 180,E1 -30950.858,E2 -30950.858} C_VEL
LIN {X 0,Y 72.172,Z 364.238,A -85,B 0,C 180,E1 -30954.411,E2 -30954.411} C_VEL
LIN {X 0,Y 72.818,Z 364.008,A -85,B 0,C 180,E1 -30959.999,E2 -30959.999} C_VEL
LIN {X 0,Y 70.412,Z 366.094,A -85,B 0,C 180,E1 -30968.607,E2 -30968.607} C_VEL
LIN {X 0,Y 67.942,Z 367.623,A -85,B 0,C 180,E1 -30970.724,E2 -30970.724} C_VEL
LIN {X 0,Y 56.763,Z 372.617,A -85,B 0,C 180,E1 -30974.336,E2 -30974.336} C_VEL
LIN {X 0,Y 44.954,Z 376.587,A -85,B 0,C 180,E1 -30980.316,E2 -30980.316} C_VEL
LIN {X 0,Y 43.584,Z 376.933,A -85,B 0,C 180,E1 -30981.246,E2 -30981.246} C_VEL
LIN {X 0,Y 38.255,Z 378.193,A -85,B 0,C 180,E1 -30984.445,E2 -30984.445} C_VEL
LIN {X 0,Y 28.839,Z 379.475,A -85,B 0,C 180,E1 -30989.337,E2 -30989.337} C_VEL
LIN {X 0,Y 21.466,Z 379.963,A -85,B 0,C 180,E1 -30996.103,E2 -30996.103} C_VEL
LIN {X 0,Y 16.807,Z 380.041,A -85,B 0,C 180,E1 -31007.127,E2 -31007.127} C_VEL
LIN {X 0,Y 15.656,Z 379.984,A -85,B 0,C 180,E1 -31012.787,E2 -31012.787} C_VEL
LIN {X 0,Y 13.41,Z 379.511,A -85,B 0,C 180,E1 -31050.044,E2 -31050.044} C_VEL
LIN {X 0,Y 14.528,Z 378.565,A -85,B 0,C 180,E1 -31078.978,E2 -31078.978} C_VEL
LIN {X 0,Y 18.413,Z 377.216,A -85,B 0,C 180,E1 -31099.811,E2 -31099.811} C_VEL
LIN {X 0,Y 26.76,Z 374.368,A -85,B 0,C 180,E1 -31116.866,E2 -31116.866} C_VEL
LIN {X 0,Y 36.334,Z 370.495,A -85,B 0,C 180,E1 -31125.334,E2 -31125.334} C_VEL
LIN {X 0,Y 46.319,Z 365.469,A -85,B 0,C 180,E1 -31130.566,E2 -31130.566} C_VEL
LIN {X 0,Y 56.578,Z 359.179,A -85,B 0,C 180,E1 -31133.676,E2 -31133.676} C_VEL
LIN {X 0,Y 58.946,Z 357.42,A -85,B 0,C 180,E1 -31134.825,E2 -31134.825} C_VEL
LIN {X 0,Y 60.337,Z 356.145,A -85,B 0,C 180,E1 -31137.04,E2 -31137.04} C_VEL
LIN {X 0,Y 60.974,Z 355.373,A -85,B 0,C 180,E1 -31140.001,E2 -31140.001} C_VEL
LIN {X 0,Y 60.758,Z 355.199,A -85,B 0,C 180,E1 -31146.643,E2 -31146.643} C_VEL
LIN {X 0,Y 60.061,Z 355.807,A -85,B 0,C 180,E1 -31151.373,E2 -31151.373} C_VEL
LIN {X 0,Y 57.82,Z 357.51,A -85,B 0,C 180,E1 -31153.451,E2 -31153.451} C_VEL
LIN {X 0,Y 47.77,Z 363.751,A -85,B 0,C 180,E1 -31156.96,E2 -31156.96} C_VEL
LIN {X 0,Y 37.89,Z 368.73,A -85,B 0,C 180,E1 -31161.921,E2 -31161.921} C_VEL
LIN {X 0,Y 28.447,Z 372.59,A -85,B 0,C 180,E1 -31170.112,E2 -31170.112} C_VEL
LIN {X 0,Y 20.012,Z 375.438,A -85,B 0,C 180,E1 -31185.34,E2 -31185.34} C_VEL
LIN {X 0,Y 15.08,Z 377.039,A -85,B 0,C 180,E1 -31208.778,E2 -31208.778} C_VEL
LIN {X 0,Y 15.039,Z 378.349,A -85,B 0,C 180,E1 -31257.816,E2 -31257.816} C_VEL
LIN {X 0,Y 18.861,Z 378.546,A -85,B 0,C 180,E1 -31278.133,E2 -31278.133} C_VEL
LIN {X 0,Y 30.104,Z 377.738,A -85,B 0,C 180,E1 -31298.983,E2 -31298.983} C_VEL
LIN {X 0,Y 36.476,Z 376.758,A -85,B 0,C 180,E1 -31304.385,E2 -31304.385} C_VEL
LIN {X 0,Y 43.087,Z 375.346,A -85,B 0,C 180,E1 -31308.076,E2 -31308.076} C_VEL
LIN {X 0,Y 55.532,Z 371.597,A -85,B 0,C 180,E1 -31312.728,E2 -31312.728} C_VEL
LIN {X 0,Y 63.502,Z 368.454,A -85,B 0,C 180,E1 -31314.81,E2 -31314.81} C_VEL
LIN {X 0,Y 65.934,Z 367.341,A -85,B 0,C 180,E1 -31316.254,E2 -31316.254} C_VEL
LIN {X 0,Y 66.133,Z 367.369,A -85,B 0,C 180,E1 -31319.999,E2 -31319.999} C_VEL
LIN {X 0,Y 63.518,Z 368.955,A -85,B 0,C 180,E1 -31325.354,E2 -31325.354} C_VEL
LIN {X 0,Y 54.444,Z 372.644,A -85,B 0,C 180,E1 -31327.416,E2 -31327.416} C_VEL
LIN {X 0,Y 43,Z 376.225,A -85,B 0,C 180,E1 -31331.364,E2 -31331.364} C_VEL
LIN {X 0,Y 36.346,Z 377.79,A -85,B 0,C 180,E1 -31334.867,E2 -31334.867} C_VEL
LIN {X 0,Y 23.787,Z 379.644,A -85,B 0,C 180,E1 -31347.633,E2 -31347.633} C_VEL
LIN {X 0,Y 15.656,Z 379.984,A -85,B 0,C 180,E1 -31372.787,E2 -31372.787} C_VEL
LIN {X 0,Y 13.668,Z 379.873,A -85,B 0,C 180,E1 -31386.006,E2 -31386.006} C_VEL
LIN {X 0,Y 11.251,Z 379.368,A -85,B 0,C 180,E1 -31411.013,E2 -31411.013} C_VEL
LIN {X 0,Y 12.034,Z 377.849,A -85,B 0,C 180,E1 -31461.329,E2 -31461.329} C_VEL
LIN {X 0,Y 17.461,Z 376.097,A -85,B 0,C 180,E1 -31484.381,E2 -31484.381} C_VEL
LIN {X 0,Y 21.025,Z 375.054,A -85,B 0,C 180,E1 -31489.328,E2 -31489.328} C_VEL
LIN {X 0,Y 31.735,Z 371.399,A -85,B 0,C 180,E1 -31495.474,E2 -31495.474} C_VEL
LIN {X 0,Y 42.19,Z 366.741,A -85,B 0,C 180,E1 -31498.642,E2 -31498.642} C_VEL
LIN {X 0,Y 52.722,Z 360.841,A -85,B 0,C 180,E1 -31500.455,E2 -31500.455} C_VEL
LIN {X 0,Y 54.956,Z 359.322,A -85,B 0,C 180,E1 -31501.978,E2 -31501.978} C_VEL
LIN {X 0,Y 54.889,Z 359.227,A -85,B 0,C 180,E1 -31505.225,E2 -31505.225} C_VEL
LIN {X 0,Y 53.134,Z 360.318,A -85,B 0,C 180,E1 -31507.16,E2 -31507.16} C_VEL
LIN {X 0,Y 42.74,Z 366.112,A -85,B 0,C 180,E1 -31509.301,E2 -31509.301} C_VEL
LIN {X 0,Y 32.429,Z 370.676,A -85,B 0,C 180,E1 -31512.696,E2 -31512.696} C_VEL
LIN {X 0,Y 22.292,Z 374.154,A -85,B 0,C 180,E1 -31518.871,E2 -31518.871} C_VEL
LIN {X 0,Y 15.783,Z 375.92,A -85,B 0,C 180,E1 -31526.969,E2 -31526.969} C_VEL
LIN {X 0,Y 9.947,Z 377.256,A -85,B 0,C 180,E1 -31544.962,E2 -31544.962} C_VEL
LIN {X 0,Y 6.705,Z 378.213,A -85,B 0,C 180,E1 -31589.912,E2 -31589.912} C_VEL
LIN {X 0,Y 9.351,Z 378.797,A -85,B 0,C 180,E1 -31638.631,E2 -31638.631} C_VEL
LIN {X 0,Y 15.069,Z 378.969,A -85,B 0,C 180,E1 -31658.761,E2 -31658.761} C_VEL
LIN {X 0,Y 28.337,Z 378.138,A -85,B 0,C 180,E1 -31672.601,E2 -31672.601} C_VEL
LIN {X 0,Y 35.232,Z 377.144,A -85,B 0,C 180,E1 -31675.623,E2 -31675.623} C_VEL
LIN {X 0,Y 42.195,Z 375.707,A -85,B 0,C 180,E1 -31677.591,E2 -31677.591} C_VEL
LIN {X 0,Y 53.035,Z 372.653,A -85,B 0,C 180,E1 -31679.999,E2 -31679.999} C_VEL
LIN {X 0,Y 42.179,Z 375.864,A -85,B 0,C 180,E1 -31681.819,E2 -31681.819} C_VEL
LIN {X 0,Y 35.198,Z 377.408,A -85,B 0,C 180,E1 -31683.583,E2 -31683.583} C_VEL
LIN {X 0,Y 21.431,Z 379.233,A -85,B 0,C 180,E1 -31690.48,E2 -31690.48} C_VEL
LIN {X 0,Y 8.999,Z 379.533,A -85,B 0,C 180,E1 -31718.756,E2 -31718.756} C_VEL
LIN {X 0,Y 6.293,Z 379.052,A -85,B 0,C 180,E1 -31770.094,E2 -31770.094} C_VEL
LIN {X 0,Y 8.99,Z 378.093,A -85,B 0,C 180,E1 -31821.53,E2 -31821.53} C_VEL
LIN {X 0,Y 14.845,Z 376.73,A -85,B 0,C 180,E1 -31841.363,E2 -31841.363} C_VEL
LIN {X 0,Y 21.025,Z 375.054,A -85,B 0,C 180,E1 -31849.328,E2 -31849.328} C_VEL
LIN {X 0,Y 23.405,Z 376.994,A -85,B 0,C 180,E1 -31851.213,E2 -31851.213} C_VEL
LIN {X 0,Y 23.405,Z 600,A -85,B 0,C 180,E1 -31851.213,E2 -31851.213} C_VEL
LIN {X 0,Y 23.405,Z 600,A -85,B 0,C 180,E1 -31851.213,E2 -31851.213}

QRS_NEXT_CUT()

QRS_NEXT()
QRS_HOME()

END
